(* Logix 5000 project; controller R1USB70001_CWRU_Scenario_Gen_20111116 vendor 1 type 14 code 54 rev 19.11; software revision 19.01; part 6 of 6 *)
(* tags used below, declared in another part *)
   ExecutePv : ExecutePv;
   ControlMode : ControlModePub;
   EditScenario : EditScenarioPub;
   Execute : ExecutePub;
   HMI : HMIPub;
   Scenario : Scenario_Def[100];
(* MainProgram, continued *)

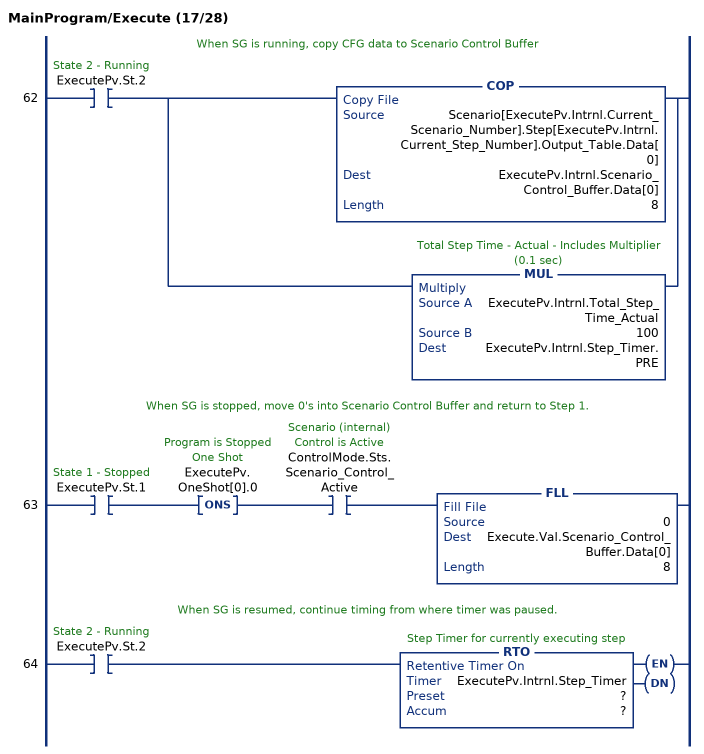
   // When SG is running, copy CFG data to Scenario Control Buffer
   62: XIC(ExecutePv.St.2)[COP(Scenario[ExecutePv.Intrnl.Current_Scenario_Number].Step[ExecutePv.Intrnl.Current_Step_Number].Output_Table.Data[0],ExecutePv.Intrnl.Scenario_Control_Buffer.Data[0],8) ,MUL(ExecutePv.Intrnl.Total_Step_Time_Actual,100,ExecutePv.Intrnl.Step_Timer.PRE) ];
   // When SG is stopped, move 0's into Scenario Control Buffer and return to Step 1.
   63: XIC(ExecutePv.St.1)ONS(ExecutePv.OneShot[0].0)XIC(ControlMode.Sts.Scenario_Control_Active)FLL(0,Execute.Val.Scenario_Control_Buffer.Data[0],8);
   // When SG is resumed, continue timing from where timer was paused.
   64: XIC(ExecutePv.St.2)RTO(ExecutePv.Intrnl.Step_Timer,?,?);
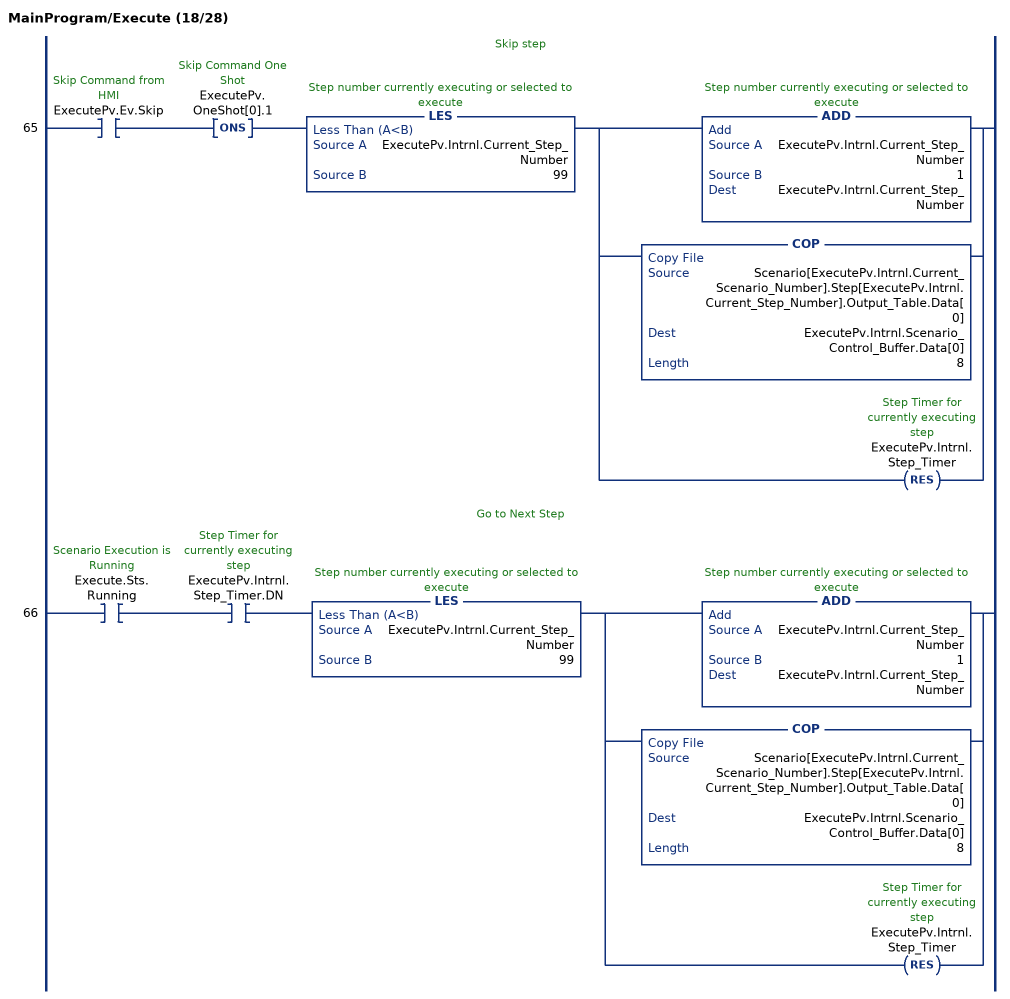
   // Skip step
   65: XIC(ExecutePv.Ev.Skip)ONS(ExecutePv.OneShot[0].1)LES(ExecutePv.Intrnl.Current_Step_Number,99)[ADD(ExecutePv.Intrnl.Current_Step_Number,1,ExecutePv.Intrnl.Current_Step_Number) ,COP(Scenario[ExecutePv.Intrnl.Current_Scenario_Number].Step[ExecutePv.Intrnl.Current_Step_Number].Output_Table.Data[0],ExecutePv.Intrnl.Scenario_Control_Buffer.Data[0],8) ,RES(ExecutePv.Intrnl.Step_Timer) ];
   // Go to Next Step
   66: XIC(Execute.Sts.Running)XIC(ExecutePv.Intrnl.Step_Timer.DN)LES(ExecutePv.Intrnl.Current_Step_Number,99)[ADD(ExecutePv.Intrnl.Current_Step_Number,1,ExecutePv.Intrnl.Current_Step_Number) ,COP(Scenario[ExecutePv.Intrnl.Current_Scenario_Number].Step[ExecutePv.Intrnl.Current_Step_Number].Output_Table.Data[0],ExecutePv.Intrnl.Scenario_Control_Buffer.Data[0],8) ,RES(ExecutePv.Intrnl.Step_Timer) ];
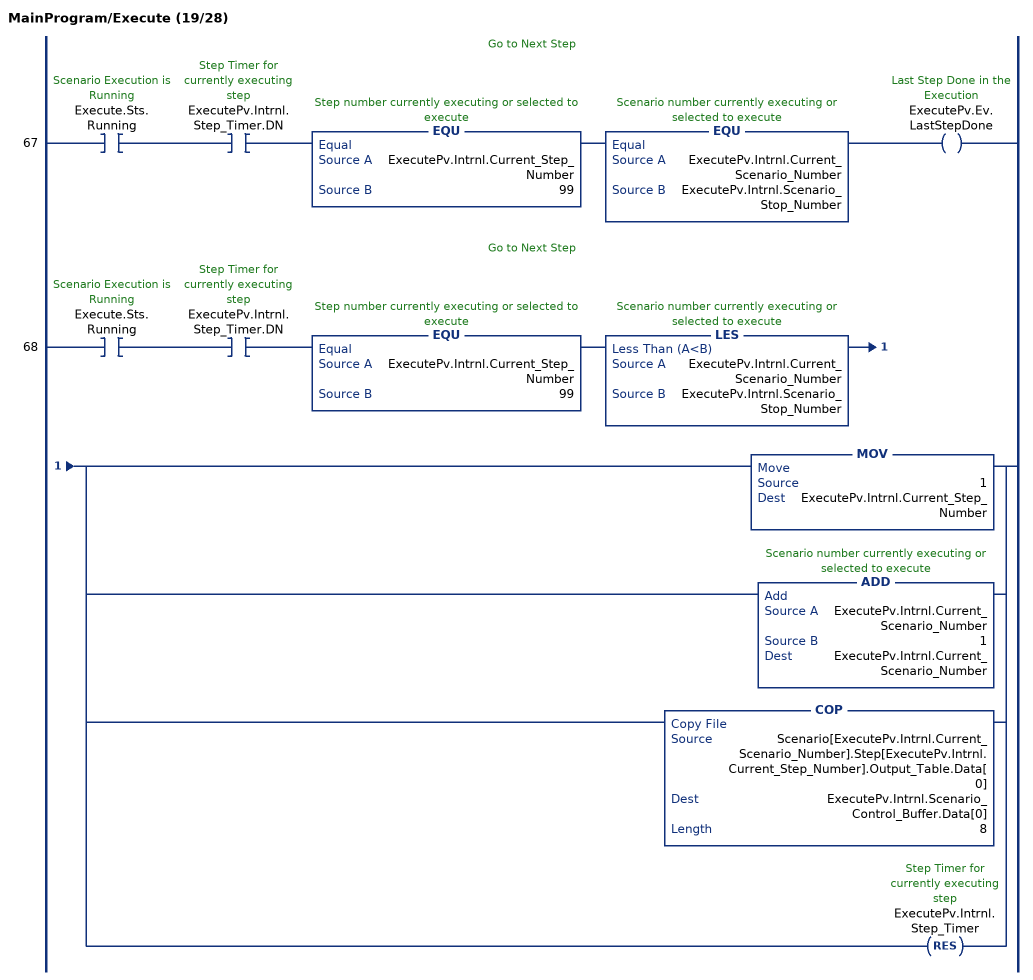
   // Go to Next Step
   67: XIC(Execute.Sts.Running)XIC(ExecutePv.Intrnl.Step_Timer.DN)EQU(ExecutePv.Intrnl.Current_Step_Number,99)EQU(ExecutePv.Intrnl.Current_Scenario_Number,ExecutePv.Intrnl.Scenario_Stop_Number)OTE(ExecutePv.Ev.LastStepDone);
   // Go to Next Step
   68: XIC(Execute.Sts.Running)XIC(ExecutePv.Intrnl.Step_Timer.DN)EQU(ExecutePv.Intrnl.Current_Step_Number,99)LES(ExecutePv.Intrnl.Current_Scenario_Number,ExecutePv.Intrnl.Scenario_Stop_Number)[MOV(1,ExecutePv.Intrnl.Current_Step_Number) ,ADD(ExecutePv.Intrnl.Current_Scenario_Number,1,ExecutePv.Intrnl.Current_Scenario_Number) ,COP(Scenario[ExecutePv.Intrnl.Current_Scenario_Number].Step[ExecutePv.Intrnl.Current_Step_Number].Output_Table.Data[0],ExecutePv.Intrnl.Scenario_Control_Buffer.Data[0],8) ,RES(ExecutePv.Intrnl.Step_Timer) ];
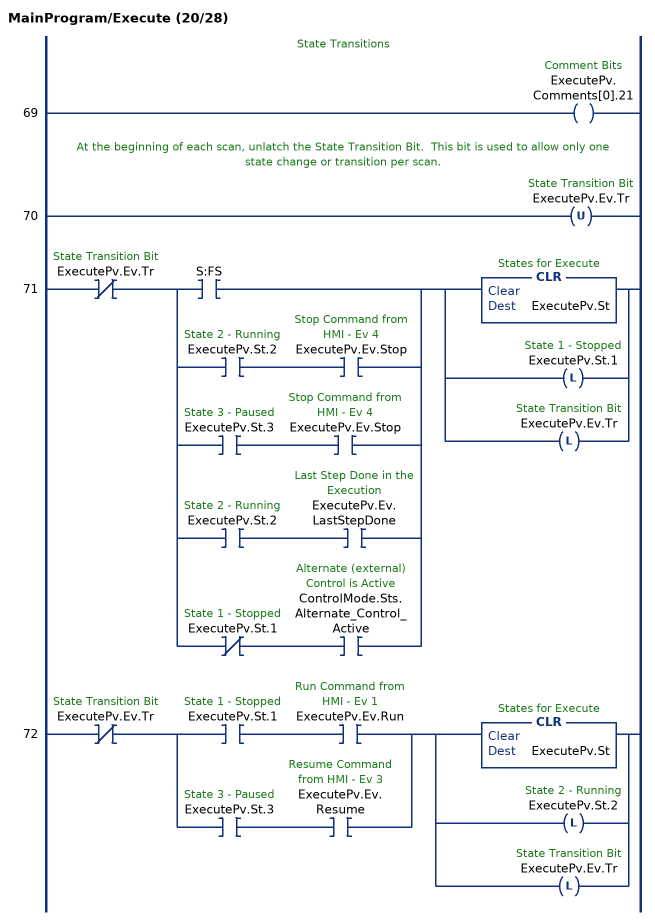
   // State Transitions
   69: OTE(ExecutePv.Comments[0].21);
   // At the beginning of each scan, unlatch the State Transition Bit.  This bit is used to allow only one state change or transition per scan.
   70: OTU(ExecutePv.Ev.Tr);
   71: XIO(ExecutePv.Ev.Tr)[XIC(S:FS) ,XIC(ExecutePv.St.2) XIC(ExecutePv.Ev.Stop) ,XIC(ExecutePv.St.3) XIC(ExecutePv.Ev.Stop) ,XIC(ExecutePv.St.2) XIC(ExecutePv.Ev.LastStepDone) ,XIO(ExecutePv.St.1) XIC(ControlMode.Sts.Alternate_Control_Active) ][CLR(ExecutePv.St) ,OTL(ExecutePv.St.1) ,OTL(ExecutePv.Ev.Tr) ];
   72: XIO(ExecutePv.Ev.Tr)[XIC(ExecutePv.St.1) XIC(ExecutePv.Ev.Run) ,XIC(ExecutePv.St.3) XIC(ExecutePv.Ev.Resume) ][CLR(ExecutePv.St) ,OTL(ExecutePv.St.2) ,OTL(ExecutePv.Ev.Tr) ];
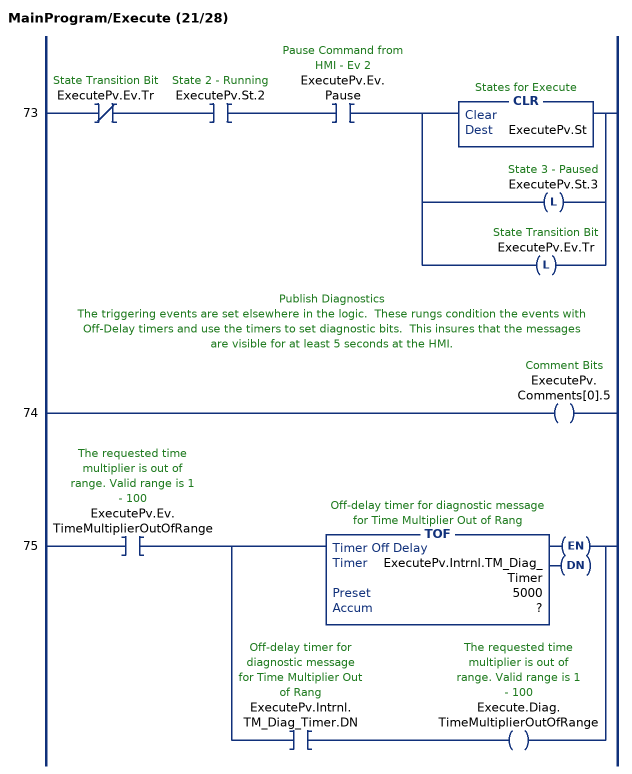
   73: XIO(ExecutePv.Ev.Tr)XIC(ExecutePv.St.2)XIC(ExecutePv.Ev.Pause)[CLR(ExecutePv.St) ,OTL(ExecutePv.St.3) ,OTL(ExecutePv.Ev.Tr) ];
   // Publish Diagnostics
   // The triggering events are set elsewhere in the logic.  These rungs condition the events with Off-Delay timers and use the timers to set diagnostic bits.  This insures that the messages are visible for at least 5 seconds at the HMI.
   74: OTE(ExecutePv.Comments[0].5);
   75: XIC(ExecutePv.Ev.TimeMultiplierOutOfRange)[TOF(ExecutePv.Intrnl.TM_Diag_Timer,?,?) ,XIC(ExecutePv.Intrnl.TM_Diag_Timer.DN) OTE(Execute.Diag.TimeMultiplierOutOfRange) ];
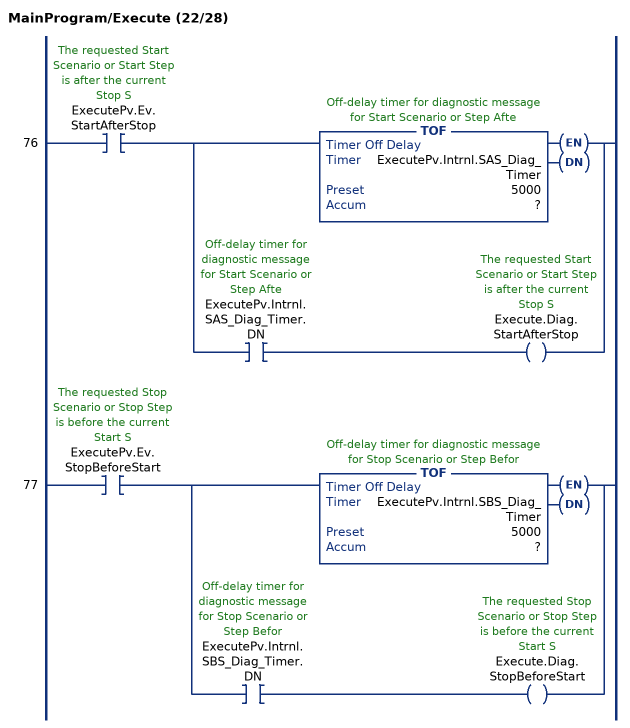
   76: XIC(ExecutePv.Ev.StartAfterStop)[TOF(ExecutePv.Intrnl.SAS_Diag_Timer,?,?) ,XIC(ExecutePv.Intrnl.SAS_Diag_Timer.DN) OTE(Execute.Diag.StartAfterStop) ];
   77: XIC(ExecutePv.Ev.StopBeforeStart)[TOF(ExecutePv.Intrnl.SBS_Diag_Timer,?,?) ,XIC(ExecutePv.Intrnl.SBS_Diag_Timer.DN) OTE(Execute.Diag.StopBeforeStart) ];
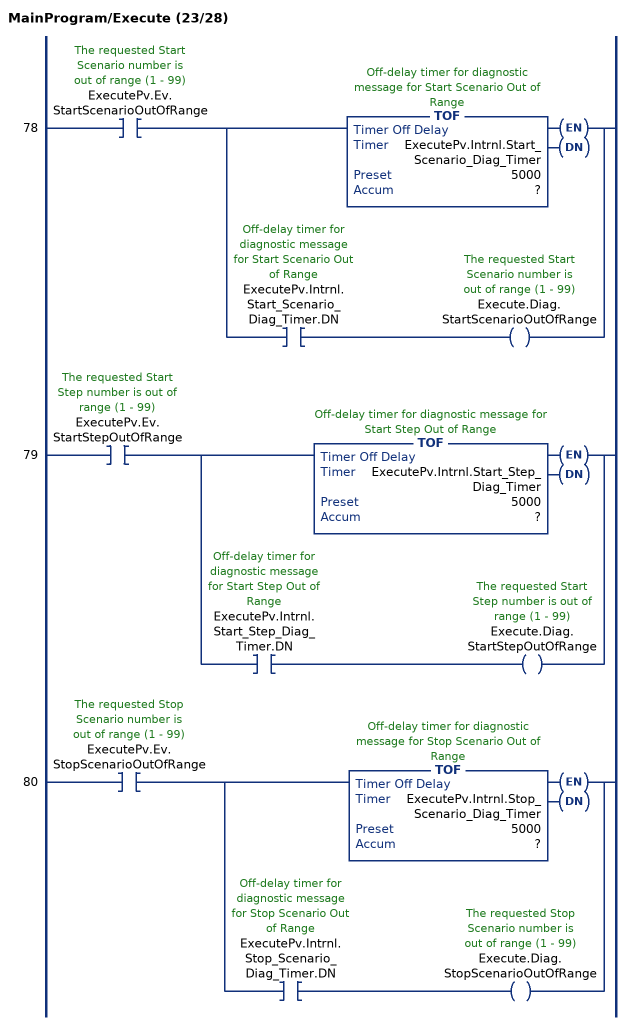
   78: XIC(ExecutePv.Ev.StartScenarioOutOfRange)[TOF(ExecutePv.Intrnl.Start_Scenario_Diag_Timer,?,?) ,XIC(ExecutePv.Intrnl.Start_Scenario_Diag_Timer.DN) OTE(Execute.Diag.StartScenarioOutOfRange) ];
   79: XIC(ExecutePv.Ev.StartStepOutOfRange)[TOF(ExecutePv.Intrnl.Start_Step_Diag_Timer,?,?) ,XIC(ExecutePv.Intrnl.Start_Step_Diag_Timer.DN) OTE(Execute.Diag.StartStepOutOfRange) ];
   80: XIC(ExecutePv.Ev.StopScenarioOutOfRange)[TOF(ExecutePv.Intrnl.Stop_Scenario_Diag_Timer,?,?) ,XIC(ExecutePv.Intrnl.Stop_Scenario_Diag_Timer.DN) OTE(Execute.Diag.StopScenarioOutOfRange) ];
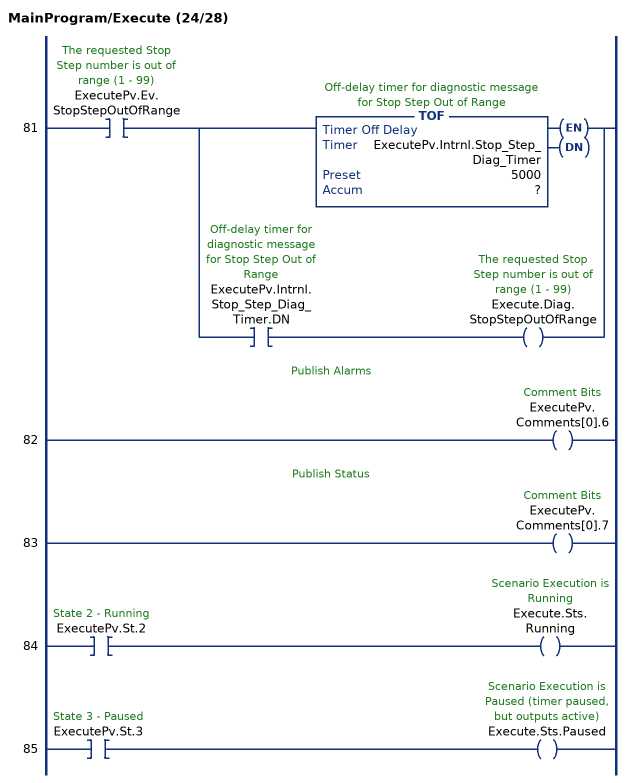
   81: XIC(ExecutePv.Ev.StopStepOutOfRange)[TOF(ExecutePv.Intrnl.Stop_Step_Diag_Timer,?,?) ,XIC(ExecutePv.Intrnl.Stop_Step_Diag_Timer.DN) OTE(Execute.Diag.StopStepOutOfRange) ];
   // Publish Alarms
   82: OTE(ExecutePv.Comments[0].6);
   // Publish Status
   83: OTE(ExecutePv.Comments[0].7);
   84: XIC(ExecutePv.St.2)OTE(Execute.Sts.Running);
   85: XIC(ExecutePv.St.3)OTE(Execute.Sts.Paused);
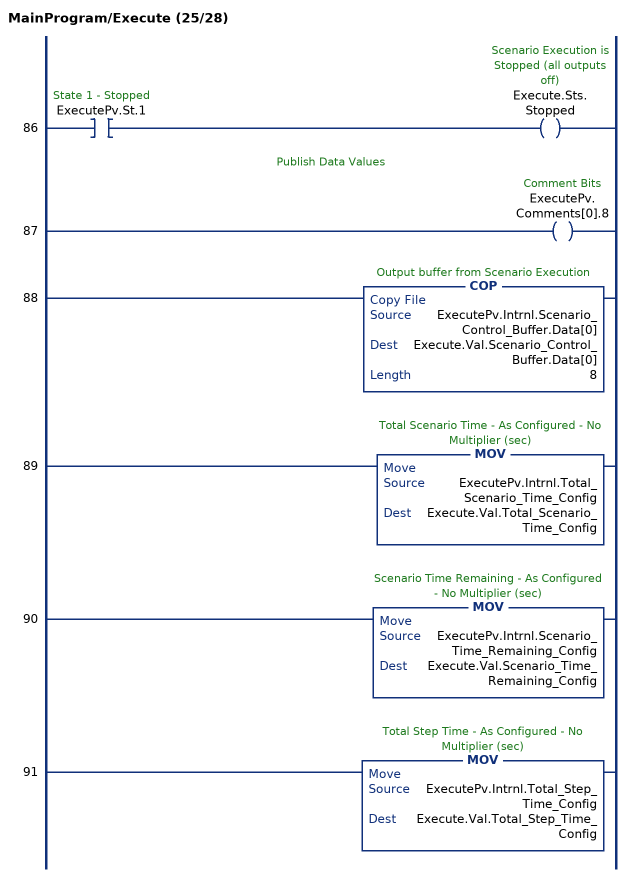
   86: XIC(ExecutePv.St.1)OTE(Execute.Sts.Stopped);
   // Publish Data Values
   87: OTE(ExecutePv.Comments[0].8);
   88: COP(ExecutePv.Intrnl.Scenario_Control_Buffer.Data[0],Execute.Val.Scenario_Control_Buffer.Data[0],8);
   89: MOV(ExecutePv.Intrnl.Total_Scenario_Time_Config,Execute.Val.Total_Scenario_Time_Config);
   90: MOV(ExecutePv.Intrnl.Scenario_Time_Remaining_Config,Execute.Val.Scenario_Time_Remaining_Config);
   91: MOV(ExecutePv.Intrnl.Total_Step_Time_Config,Execute.Val.Total_Step_Time_Config);
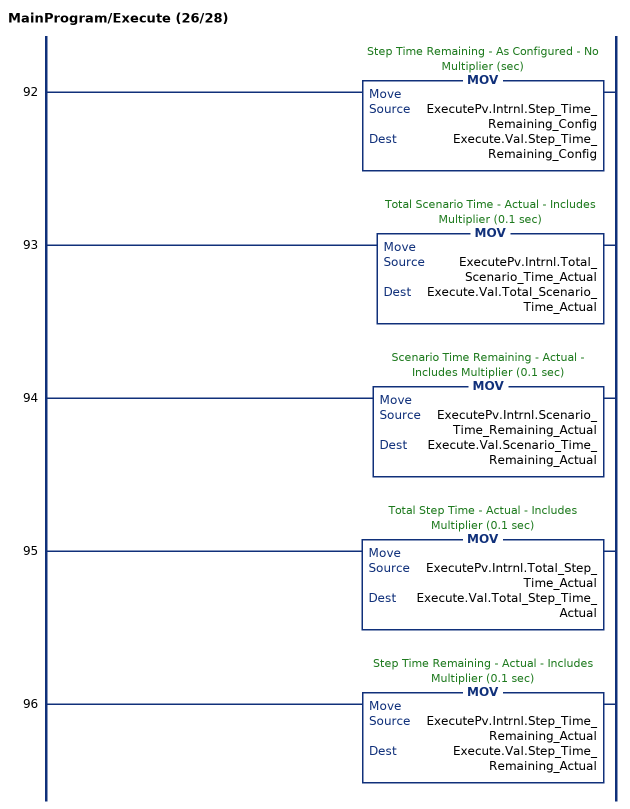
   92: MOV(ExecutePv.Intrnl.Step_Time_Remaining_Config,Execute.Val.Step_Time_Remaining_Config);
   93: MOV(ExecutePv.Intrnl.Total_Scenario_Time_Actual,Execute.Val.Total_Scenario_Time_Actual);
   94: MOV(ExecutePv.Intrnl.Scenario_Time_Remaining_Actual,Execute.Val.Scenario_Time_Remaining_Actual);
   95: MOV(ExecutePv.Intrnl.Total_Step_Time_Actual,Execute.Val.Total_Step_Time_Actual);
   96: MOV(ExecutePv.Intrnl.Step_Time_Remaining_Actual,Execute.Val.Step_Time_Remaining_Actual);
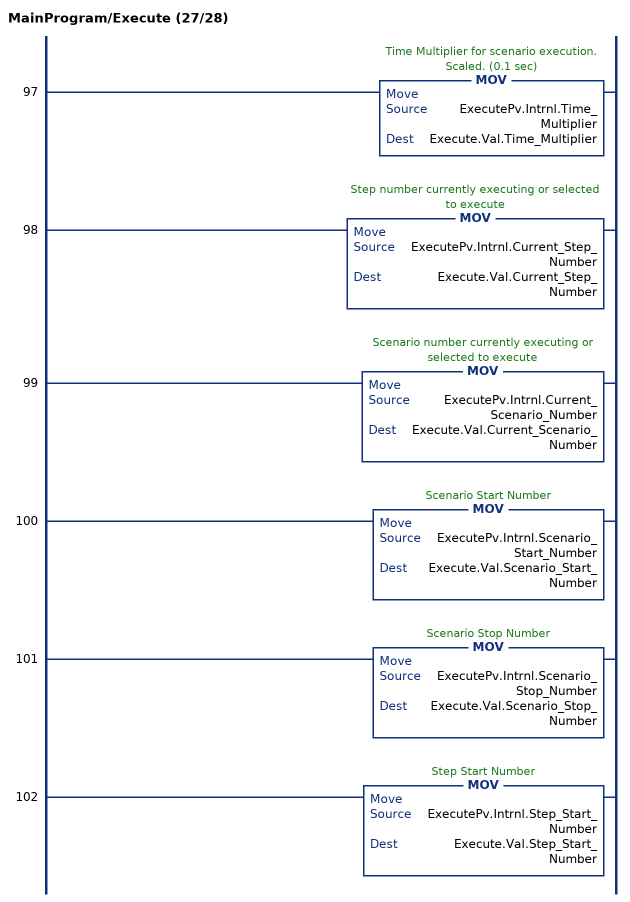
   97: MOV(ExecutePv.Intrnl.Time_Multiplier,Execute.Val.Time_Multiplier);
   98: MOV(ExecutePv.Intrnl.Current_Step_Number,Execute.Val.Current_Step_Number);
   99: MOV(ExecutePv.Intrnl.Current_Scenario_Number,Execute.Val.Current_Scenario_Number);
   100: MOV(ExecutePv.Intrnl.Scenario_Start_Number,Execute.Val.Scenario_Start_Number);
   101: MOV(ExecutePv.Intrnl.Scenario_Stop_Number,Execute.Val.Scenario_Stop_Number);
   102: MOV(ExecutePv.Intrnl.Step_Start_Number,Execute.Val.Step_Start_Number);
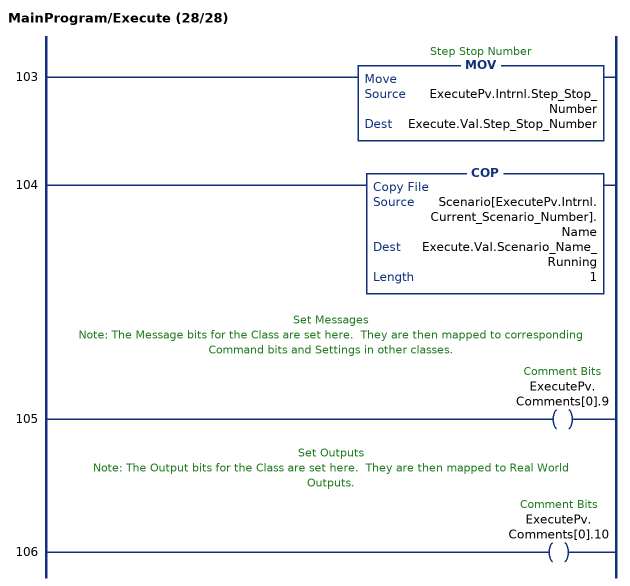
   103: MOV(ExecutePv.Intrnl.Step_Stop_Number,Execute.Val.Step_Stop_Number);
   104: COP(Scenario[ExecutePv.Intrnl.Current_Scenario_Number].Name,Execute.Val.Scenario_Name_Running,1);
   // Set Messages
   // Note: The Message bits for the Class are set here.  They are then mapped to corresponding Command bits and Settings in other classes.
   105: OTE(ExecutePv.Comments[0].9);
   // Set Outputs
   // Note: The Output bits for the Class are set here.  They are then mapped to Real World Outputs.
   106: OTE(ExecutePv.Comments[0].10);
END_ROUTINE

ROUTINE MainRoutine   (* ladder *)
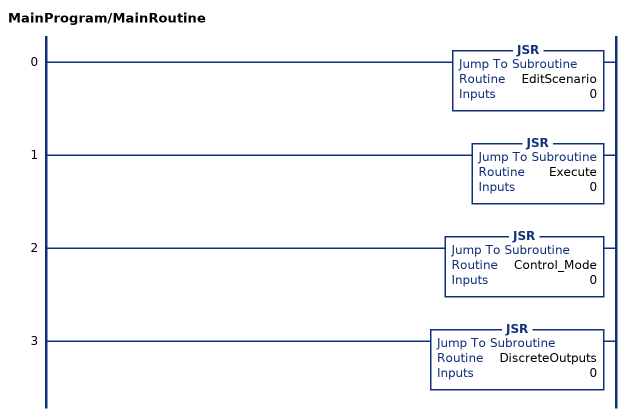
   0: JSR(EditScenario,0);
   1: JSR(Execute,0);
   2: JSR(Control_Mode,0);
   3: JSR(DiscreteOutputs,0);
END_ROUTINE
END_PROGRAM
